// TIA Portal V17 export
// export: Created 2025-04-09T08:03:05.7421914Z, ExportSetting WithDefaults, DisplayName Totally Integrated Automation Portal, DisplayVersion V17 Update 8, DisplayName TIA Portal Openness, DisplayVersion V17 Update 8, DisplayName TIA Portal Version Control Interface, DisplayVersion V17, DisplayName SINAMICS Startdrive Advanced, DisplayVersion V17 SP2, DisplayName SINAMICS Startdrive G110M, G120, G120C, G120D, G120P, G115D, DisplayVersion V17 SP2, DisplayName SINAMICS Startdrive G130, G150, S120, S150, SINAMICS MV, S210, DisplayVersion V17 SP2, DisplayName STEP 7 Professional, DisplayVersion V17 Update 8, DisplayName SINUMERIK ONE STEP 7 Toolbox, DisplayVersion V17 Update 12, DisplayName SINUMERIK ONE PLC Basic Program Plus, DisplayVersion V17 Update 12, DisplayName SINUMERIK 840D sl STEP 7 Toolbox, DisplayVersion V17 Update 12, DisplayName STEP 7 Safety, DisplayVersion V17 Update 6, DisplayName WinCC Advanced, DisplayVersion V17 Update 8
FUNCTION "FC2003_CNC_MODES" : Void   // FC2003, LAD
{ S7_Optimized_Access := 'FALSE' }
AUTHOR : ETXETAR
VERSION : 1.0
// stored: AutoNumber false, IsIECCheckEnabled false, SetENOAutomatically false, UDAEnableTagReadback false
   VAR CONSTANT
      FC_NUMBER : DInt := 2003;
   END_VAR
BEGIN

REGION Network 1: CNC MODES MODE GROUP 1
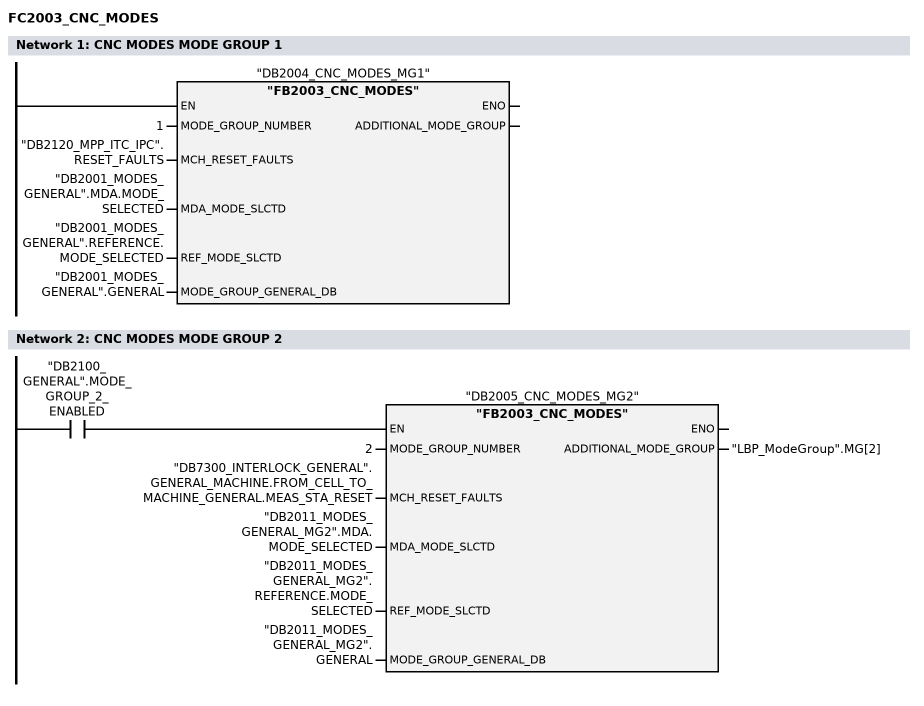
   RUNG wire#powerrail
      "DB2004_CNC_MODES_MG1"(MODE_GROUP_NUMBER := 1, MCH_RESET_FAULTS := "DB2120_MPP_ITC_IPC".RESET_FAULTS, MDA_MODE_SLCTD := "DB2001_MODES_GENERAL".MDA.MODE_SELECTED, REF_MODE_SLCTD := "DB2001_MODES_GENERAL".REFERENCE.MODE_SELECTED, MODE_GROUP_GENERAL_DB := "DB2001_MODES_GENERAL".GENERAL, ADDITIONAL_MODE_GROUP =>)
   END_RUNG
   // the same network as SCL:
   "DB2004_CNC_MODES_MG1"(MODE_GROUP_NUMBER := 1,   // "FB2003_CNC_MODES"
                          MCH_RESET_FAULTS := "DB2120_MPP_ITC_IPC".RESET_FAULTS,
                          MDA_MODE_SLCTD := "DB2001_MODES_GENERAL".MDA.MODE_SELECTED,
                          REF_MODE_SLCTD := "DB2001_MODES_GENERAL".REFERENCE.MODE_SELECTED,
                          MODE_GROUP_GENERAL_DB := "DB2001_MODES_GENERAL".GENERAL);
END_REGION

REGION Network 2: CNC MODES MODE GROUP 2
   RUNG wire#powerrail
      Contact( "DB2100_GENERAL".MODE_GROUP_2_ENABLED )
      "DB2005_CNC_MODES_MG2"(MODE_GROUP_NUMBER := 2, MCH_RESET_FAULTS := "DB7300_INTERLOCK_GENERAL".GENERAL_MACHINE.FROM_CELL_TO_MACHINE_GENERAL.MEAS_STA_RESET, MDA_MODE_SLCTD := "DB2011_MODES_GENERAL_MG2".MDA.MODE_SELECTED, REF_MODE_SLCTD := "DB2011_MODES_GENERAL_MG2".REFERENCE.MODE_SELECTED, MODE_GROUP_GENERAL_DB := "DB2011_MODES_GENERAL_MG2".GENERAL, ADDITIONAL_MODE_GROUP => "LBP_ModeGroup".MG[2])
   END_RUNG
   // the same network as SCL:
   IF "DB2100_GENERAL".MODE_GROUP_2_ENABLED THEN
       "DB2005_CNC_MODES_MG2"(MODE_GROUP_NUMBER := 2,   // "FB2003_CNC_MODES"
                              MCH_RESET_FAULTS := "DB7300_INTERLOCK_GENERAL".GENERAL_MACHINE.FROM_CELL_TO_MACHINE_GENERAL.MEAS_STA_RESET,
                              MDA_MODE_SLCTD := "DB2011_MODES_GENERAL_MG2".MDA.MODE_SELECTED,
                              REF_MODE_SLCTD := "DB2011_MODES_GENERAL_MG2".REFERENCE.MODE_SELECTED,
                              MODE_GROUP_GENERAL_DB := "DB2011_MODES_GENERAL_MG2".GENERAL,
                              ADDITIONAL_MODE_GROUP => "LBP_ModeGroup".MG[2]);
   END_IF;
END_REGION
END_FUNCTION
